PROGRAM P_Demo_PLC_ReadSymInfoByName
VAR
    fbPLC_ReadSymInfoByName : PLC_ReadSymInfoByName; // PLC_ReadSymInfoByName 实例
    NETID                   : T_AmsNetId;
    PORT                    : T_AmsPort;
    SYMNAME                 : T_MaxString;
    START                   : BOOL;
    TMOUT                   : TIME := DEFAULT_ADS_TIMEOUT;
    BUSY                    : BOOL;
    ERR                     : BOOL;
    ERRID                   : UDINT;
    SymInfo                 : SYMINFOSTRUCT;
END_VAR

// =============================================================================
// 场景：按名查变量。
// 价值：O(1)。
// 验证：给变量名，读出对应符号信息。
// 验证步骤：
//   1. 右键 PLC 项目下 POUs 文件夹 → Add → Existing Item → 选本 .TcPOU 文件
//   2. 引用 Tc2_Utilities（References → Add library）
//   3. 编译 → 登录 → 运行；按上方『验证』行的指示在线写值观察
// =============================================================================

// 单次完整调用形式（所有 VAR_INPUT 显式赋值）
fbPLC_ReadSymInfoByName(
    NETID := NETID,
    PORT := PORT,
    SYMNAME := SYMNAME,
    START := START,
    TMOUT := TMOUT,
    BUSY => BUSY,
    ERR => ERR,
    ERRID => ERRID,
    SymInfo => SymInfo
);

END_PROGRAM

(* stored: Version 1.1.0.1, ProductVersion 3.1.4024.5
   POU P_Demo_PLC_ReadSymInfoByName: Id {8a50c1f9-959e-5ade-8404-73aed60dbc42}, SpecialFunc None *)
